FUNCTION_BLOCK Q_ChildLocation (* Command change child location ( Part 6 - F.14 ) *)
  (* Standard: ISO 11783-6; Description: Copyright (c) 2022 HR Agrartechnik GmbH This program and the accompanying materials are made available under the terms of the Eclipse Public License 2.0 which is available at https://www.eclipse.org/legal/epl-2.0/ SPDX-License-Identifier: EPL-2.0 see Description Tab *)
  (* Version 1.0, 2022-07-08, Franz Höpfinger, HR Agrartechnik GmbH *)
  PACKAGE isobus::UT::Q;
  IMPORT isobus::UT::Q::const::IDs::ID_NULL;
  (* Documentation:
  Command change child location ( Part 6 - F.14 )
   The Change Child Location command is used to change the relative position of an object. The command addresses two distinct Object IDs with different validity rules each — u16ObjId (the child object to move) and u16ObjIdParent (the parent it is moved within). Annex F only defines which object types are valid as the child; which object types may act as parent for this command is defined separately in Annex B, under each object type's "Allowed commands" list.
   Valid values for u16ObjId (the child object to move)
   Valid if it falls within one of the following ISO 11783-6 ID ranges (Annex F.14):
    - Container: 3000 – 3999
   - Key: 5000 – 5999
   - Button: 6000 – 6999
   - InputBooleanField: 7000 – 7999
   - InputStringField: 8000 – 8999
   - InputNumberField: 9000 – 9999
   - InputListField: 10000 – 10999
   - OutputStringField: 11000 – 11999
   - OutputNumberField: 12000 – 12999
   - TypLine: 13000 – 13999
   - TypRectangle: 14000 – 14999
   - TypEllipse: 15000 – 15999
   - TypPolygon: 16000 – 16999
   - Meter: 17000 – 17999
   - LinearBarGraph: 18000 – 18999
   - ArchedBarGraph: 19000 – 19999
   - PictureGraphic: 20000 – 20499
   - ObjectPointer: 27000 – 27999
   - OutputListObject: 37000 – 37999
   - ExternalObjectPointer: 43000 – 43999
   - AnimationObject: 44000 – 44999
   - ScaledGraphicObject: 48000 – 48999
   - AuxiliaryFunction: 29000 – 29999
   - AuxiliaryFunctionType2: 31000 – 31999
   - AuxiliaryInput: 30000 – 30999
   - AuxiliaryInputType2: 32000 – 32999
   - AuxiliaryControlDesignator: 33000 – 33999
    Valid values for u16ObjIdParent (the parent object)
   Only object types whose ISO 11783-6 Annex B definition lists "Change Child Location command" / "Change Child Position command" among its Allowed commands:
    - WorkingSet (Annex B.1)
   - DataMask (Annex B.2)
   - AlarmMask (Annex B.3)
   - Container (Annex B.4)
   - Key (Annex B.6)
   - WindowMask
   - Button
   - AuxiliaryFunction / AuxiliaryFunctionType2
   - AuxiliaryInput / AuxiliaryInputType2
    Not valid as parent: SoftKeyMask (Annex B.5 does not list either command as allowed) and AnimationObject (its children are indexed frames, not X/Y-positioned).
   ID_NULL (65535) is not a command target but can be used in INIT to deactivate the FB. Any child ID outside the child ranges above, or any parent ID that is not one of the parent-capable types above, is invalid for commanding — independent of each other.
   Activate / Deactivate
   The FB is deactivated by default. It becomes active when INIT provides a valid child location Object ID. Sending INIT with ID_NULL (65535) deactivates the FB again. This toggle can be repeated arbitrarily.
    - INIT + ID_NULL (65535): FB deactivated, STATUS="DEACTIVATED", s16result=VT_E_DEACTIVATED (-40)
   - INIT + valid child location ID: FB activated, STATUS="initialized", s16result=VT_E_NO_ERR (0). If a REQ was buffered before, it is executed immediately.
   - INIT + invalid ID: STATUS="ERROR: Invalid Object ID (not a child location object)", s16result=VT_E_INVALID_OBJECT_ID (-132)
    REQ Handling
    - REQ before any INIT: Buffered, STATUS="Buffered: INIT not yet completed", s16result=VT_E_NOT_READY (-131)
   - REQ while deactivated (INIT came with NULL or invalid ID): STATUS shows the actual deactivation reason, s16result=VT_E_DEACTIVATED (-40) or VT_E_INVALID_OBJECT_ID (-132)
   - REQ while active: Command sent to VT, result reflected in CNF
    param[in] {objectID, uint16_t}
   Object ID. Use ID_NULL (65535) to deactivate the FB. Use a valid child location object ID to activate.
   param[in] {parentObjectID, uint16_t}
   Parent object ID
   param[in] {relativeXPositionChange, uint8_t}
   Relative change in x position (interpreted as signed!)
   param[in] {relativeYPositionChange, uint8_t}
   Relative change in y position (interpreted as signed!)
   Return Values (s16result):
   int16_t
    - VT_E_NO_ERR (0) - OK
   - VT_E_DEACTIVATED (-40) - FB deactivated (INIT received with ID_NULL)
   - VT_E_INVALID_OBJECT_ID (-132) - Object ID is invalid (not a child location object)
   - VT_E_NOT_READY (-131) - Buffered: INIT not yet completed
   - VT_E_OVERFLOW (-6) - buffer overflow
   - VT_E_NOACT (-8) - Command not possible in current state
   - VT_E_NO_INSTANCE (-21) - No VT client available
   - VT_E_ISO_INSTANCE_INVALID (-129) - Identifier for instance (connection) invalid
   - VT_E_NOT_ALIVE (-130) - Identifier for instance valid, but VT Dead.
  *)
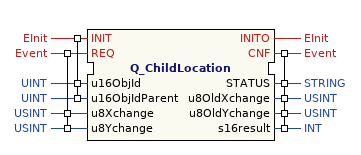
  EVENT_INPUT
    INIT : EInit WITH u16ObjId, u16ObjIdParent; (* Service Initialization *)
    REQ WITH u8Xchange, u8Ychange; (* Service Request *)
  END_EVENT
  EVENT_OUTPUT
    INITO : EInit; (* Initialization Confirm *)
    CNF WITH STATUS, u8OldYchange, u8OldXchange, s16result; (* Confirmation of Requested Service *)
  END_EVENT
  VAR_INPUT
    u16ObjId : UINT := ID_NULL; (* Object ID *)
    u16ObjIdParent : UINT := ID_NULL; (* Parent object ID *)
    u8Xchange : USINT; (* Relative change in x position (interpreted as signed!) *)
    u8Ychange : USINT; (* Relative change in y position (interpreted as signed!) *)
  END_VAR
  VAR_OUTPUT
    STATUS : STRING; (* Service Status *)
    u8OldXchange : USINT; (* Old relative change in x position (interpreted as signed!) *)
    u8OldYchange : USINT; (* Old relative change in y position (interpreted as signed!) *)
    s16result : INT; (* retval see description *)
  END_VAR
END_FUNCTION_BLOCK
